FUNCTION_BLOCK EL3012
VAR
	_io : EL3xx2_Data;
	{attribute addProperty Name "WcState"}
	_wcState : WcStateInputToggle;
	{attribute addProperty Name "Info data"}
	_infoData : InfoDataAds;
END_VAR

PROPERTY IO : REFERENCE TO EL3xx2_Data
GET
IO REF= _io;
END_GET
END_PROPERTY

PROPERTY WcState : REFERENCE TO WcStateInputToggle
GET
WcState REF= _wcState;
END_GET
END_PROPERTY

END_FUNCTION_BLOCK

(* stored: Version 1.1.0.1, ProductVersion 3.1.4024.9
   POU EL3012: Id {e16b901d-dfc8-0762-0ee9-7f258bee590d}, SpecialFunc None
   Property IO: Id {64bb6a81-22d2-01ff-2582-0be9f69d74a3}
   Get Get: Id {0d04b8e3-4134-0f32-110a-a360122d03da}
   Property WcState: Id {f91c4bed-c77f-0a84-3d7e-e2e5a71aaec6}
   Get Get: Id {e0a841cf-af6d-01c8-2fd4-f8448dc9671b} *)
